TYPE ServoMotion_FunctionResult :
(
	MOTION_OK := -1,
	MOTION_BUSY := 0,
	MOTION_UNKNOWN_AXIS,
	MOTION_UNKNOWN_AXIS_GROUP,
	MOTION_UNKNOWN_SAME_AXIS_IN_GROUP,
	MOTION_COMMAND_ABORTED,
	MOTION_ERROR
);
END_TYPE

(* stored: Version 1.1.0.1, ProductVersion 3.1.0.36
   DUT ServoMotion_FunctionResult: Id {911881e7-7e36-422a-bfa6-aaaacebbd843} *)
